// TIA Portal V16 export
// export: Created 2022-02-04T14:40:10.8066847Z, ExportSetting WithDefaults, DisplayName Totally Integrated Automation Portal, DisplayVersion V16 Update 1, DisplayName TIA Portal Version Control Interface, DisplayVersion V16, DisplayName TIA Portal Openness, DisplayVersion V16, DisplayName SINAMICS Startdrive Advanced, DisplayVersion V16 Update 5, DisplayName SINAMICS Startdrive G130, G150, S120, S150, SINAMICS MV, S210, DisplayVersion V16 Update 5, DisplayName SINAMICS Startdrive G110M, G120, G120C, G120D, G120P, G115D, DisplayVersion V16 Update 5, DisplayName STEP 7 Professional, DisplayVersion V16, DisplayName STEP 7 Safety, DisplayVersion V16, DisplayName WinCC Advanced, DisplayVersion V16, DisplayName SIMATIC Visualization Architect, DisplayVersion V16
FUNCTION_BLOCK "ПФМ Брака"   // FB3, LAD
VERSION : 0.1
// логика работы ПФМ брака
// stored: AutoNumber true, IsIECCheckEnabled false, UDAEnableTagReadback false
   VAR DB_SPECIFIC
      Trig332 : Bool;   // Тригер М332 сброс доски
      "TrigS79.3" : Bool;   // Тригер Авто режима
      ForcingPacket : Bool;
      LiftPushingPacket : Bool;   // лифт занят
      HodVil2 { ExternalAccessible := 'False'; ExternalVisible := 'False'; ExternalWritable := 'False'} : Bool;   // Триггер ход вил М335
      HodVil { ExternalAccessible := 'False'; ExternalVisible := 'False'; ExternalWritable := 'False'} : Bool;   // Триггер ход вил М335
      ForcingLift : Bool;
      CountSensor_front : Bool;
      StopDovod : Bool;
      StopDropppingBoards : Bool;
      newBob_old : Bool;
      liftDown_old : Bool;
      liftPushingPacket_old : Bool;
      newBoard_old : Bool;
      Upor_Off_trig : Bool;
      Lift_GoToStartPosition : Bool;
      ReviveSignal : Bool;   // сигнал для оживления механизмов
      StartAwaitForGasket : Bool;   // ожидание прокладок
      AwaitGasket : Bool;
      AlarmNotReadedPack : Bool;
      AlarmExtraBoardInLay : Bool;   // авария лишняя доска на слой ПФМ брака
      AlarmNoPacketPushed : Bool;
      BoardsInLayCounter : Int;   // Сравнение счетчика 2
      LayersCounter : Int;   // Счет слоев досок
   END_VAR
   VAR
      Board_counter : "Adder";   // Счетчик досок в слое
      Lay_counter : "Adder";   // Счетчик слоев
   END_VAR
   VAR_TEMP
      start_await : Bool;
      Sert : Word;
   END_VAR
   VAR_TEMP   // added for the SCL form of the ladder/FBD networks
      _w1 : Bool;
      _w2 : Bool;
      _w3 : Bool;
      _s5time1 : S5Time;
   END_VAR
BEGIN

REGION Network 1: Реле безопасности К41 группа 331,332-337
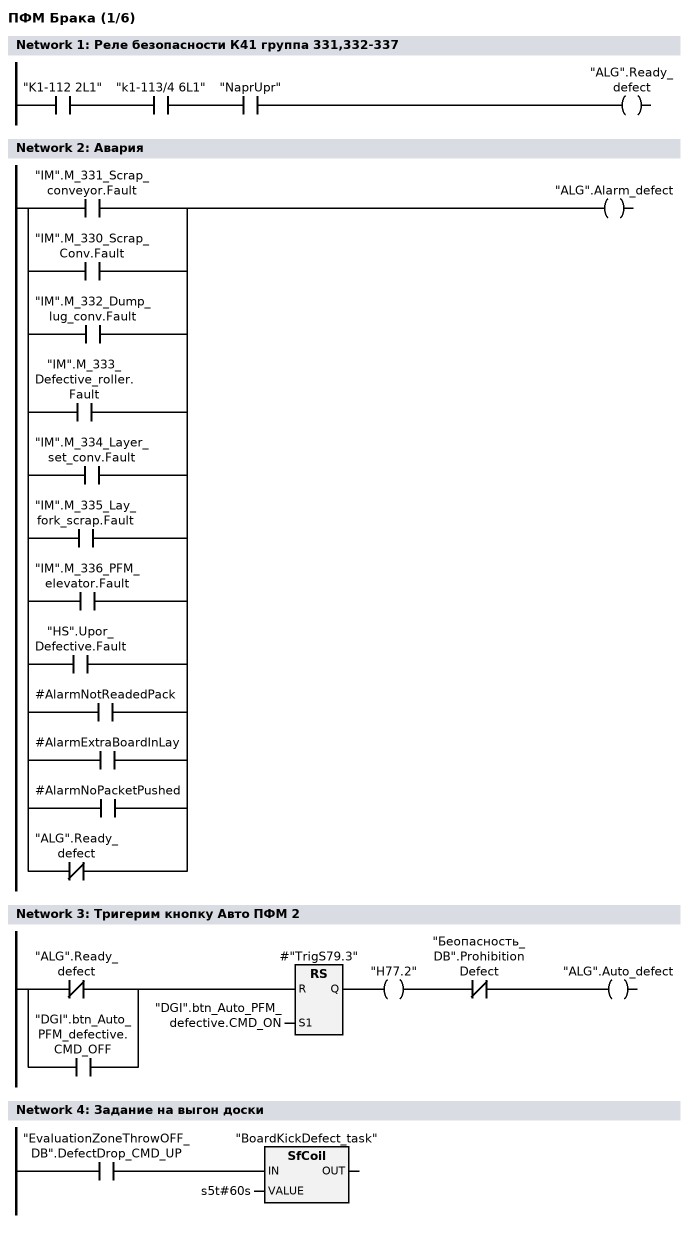
   RUNG wire#powerrail
      Contact( "K1-112 2L1" )
      Contact( "k1-113/4 6L1" )
      Contact( "NaprUpr" )
      Coil( "ALG".Ready_defect )
   END_RUNG
   // the same network as SCL:
   "ALG".Ready_defect := "K1-112 2L1" AND "k1-113/4 6L1" AND "NaprUpr";
END_REGION

REGION Network 2: Авария
   RUNG wire#powerrail
      Contact( "IM".M_331_Scrap_conveyor.Fault )
      wire#w1
      Coil( "ALG".Alarm_defect )
   END_RUNG
   RUNG wire#powerrail
      Contact( "IM".M_330_Scrap_Conv.Fault )
   END_RUNG wire#w1
   RUNG wire#powerrail
      Contact( "IM".M_332_Dump_lug_conv.Fault )
   END_RUNG wire#w1
   RUNG wire#powerrail
      Contact( "IM".M_333_Defective_roller.Fault )
   END_RUNG wire#w1
   RUNG wire#powerrail
      Contact( "IM".M_334_Layer_set_conv.Fault )
   END_RUNG wire#w1
   RUNG wire#powerrail
      Contact( "IM".M_335_Lay_fork_scrap.Fault )
   END_RUNG wire#w1
   RUNG wire#powerrail
      Contact( "IM".M_336_PFM_elevator.Fault )
   END_RUNG wire#w1
   RUNG wire#powerrail
      Contact( "HS".Upor_Defective.Fault )
   END_RUNG wire#w1
   RUNG wire#powerrail
      Contact( #AlarmNotReadedPack )
   END_RUNG wire#w1
   RUNG wire#powerrail
      Contact( #AlarmExtraBoardInLay )
   END_RUNG wire#w1
   RUNG wire#powerrail
      Contact( #AlarmNoPacketPushed )
   END_RUNG wire#w1
   RUNG wire#powerrail
      I_Contact( "ALG".Ready_defect )
   END_RUNG wire#w1
   // the same network as SCL:
   "ALG".Alarm_defect := "IM".M_331_Scrap_conveyor.Fault OR "IM".M_330_Scrap_Conv.Fault OR "IM".M_332_Dump_lug_conv.Fault OR "IM".M_333_Defective_roller.Fault OR "IM".M_334_Layer_set_conv.Fault OR "IM".M_335_Lay_fork_scrap.Fault OR "IM".M_336_PFM_elevator.Fault OR "HS".Upor_Defective.Fault OR #AlarmNotReadedPack OR #AlarmExtraBoardInLay OR #AlarmNoPacketPushed OR NOT "ALG".Ready_defect;
END_REGION

REGION Network 3: Тригерим кнопку Авто ПФМ 2
   RUNG wire#powerrail
      I_Contact( "ALG".Ready_defect )
      wire#w1
      S_RS(operand := #"TrigS79.3", s1 := "DGI".btn_Auto_PFM_defective.CMD_ON)
      Coil( "H77.2" )
      I_Contact( "Беопасность_DB".ProhibitionDefect )
      Coil( "ALG".Auto_defect )
   END_RUNG
   RUNG wire#powerrail
      Contact( "DGI".btn_Auto_PFM_defective.CMD_OFF )
   END_RUNG wire#w1
   // the same network as SCL:
   IF NOT "ALG".Ready_defect OR "DGI".btn_Auto_PFM_defective.CMD_OFF THEN
       #"TrigS79.3" := FALSE;   // RS flip-flop
   END_IF;
   IF "DGI".btn_Auto_PFM_defective.CMD_ON THEN #"TrigS79.3" := TRUE; END_IF;
   "H77.2" := #"TrigS79.3";
   "ALG".Auto_defect := #"TrigS79.3" AND NOT "Беопасность_DB".ProhibitionDefect;
END_REGION

REGION Network 4: Задание на выгон доски
   // no SCL statement known for SfCoil: written as a call
   SfCoil(in := "EvaluationZoneThrowOFF_DB".DefectDrop_CMD_UP,
          value := s5t#60s,
          operand := "BoardKickDefect_task");
END_REGION

REGION Network 5: Авто вперед М331/ M330
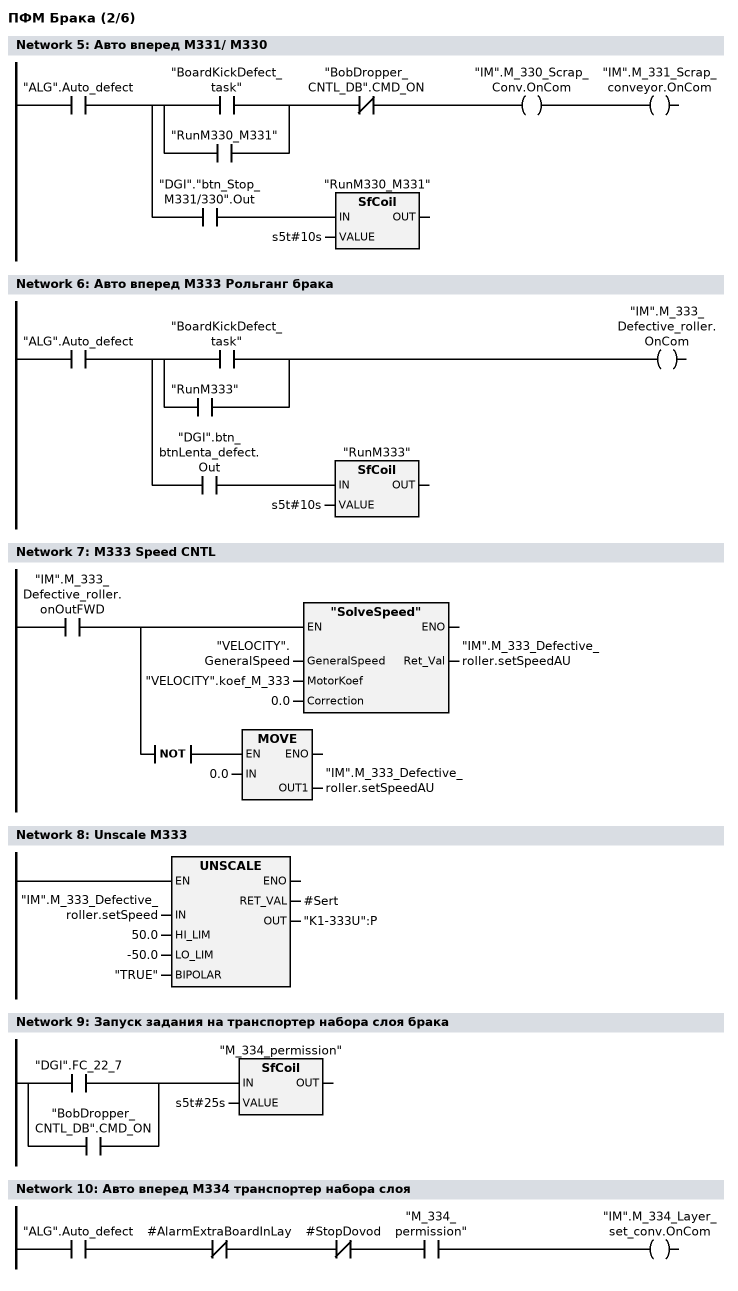
   // no SCL statement known for SfCoil: written as a call
   "IM".M_330_Scrap_Conv.OnCom := "ALG".Auto_defect AND ("BoardKickDefect_task" OR "RunM330_M331") AND NOT "BobDropper_CNTL_DB".CMD_ON;
   "IM".M_331_Scrap_conveyor.OnCom := "IM".M_330_Scrap_Conv.OnCom;
   SfCoil(in := "ALG".Auto_defect AND "DGI"."btn_Stop_M331/330".Out,
          value := s5t#10s,
          operand := "RunM330_M331");
END_REGION

REGION Network 6: Авто вперед М333 Рольганг брака
   // no SCL statement known for SfCoil: written as a call
   "IM".M_333_Defective_roller.OnCom := "ALG".Auto_defect AND ("BoardKickDefect_task" OR "RunM333");
   SfCoil(in := "ALG".Auto_defect AND "DGI".btn_btnLenta_defect.Out, value := s5t#10s, operand := "RunM333");
END_REGION

REGION Network 7: М333 Speed CNTL
   RUNG wire#powerrail
      Contact( "IM".M_333_Defective_roller.onOutFWD )
      wire#w1
      "SolveSpeed"(GeneralSpeed := "VELOCITY".GeneralSpeed, MotorKoef := "VELOCITY".koef_M_333, Correction := 0.0, Ret_Val => "IM".M_333_Defective_roller.setSpeedAU)
   END_RUNG
   RUNG wire#w1
      Not()
      { S7_GenerateENO := "TRUE" } Move(in := 0.0, out1 => "IM".M_333_Defective_roller.setSpeedAU)
   END_RUNG
   // the same network as SCL:
   #_w1 := "IM".M_333_Defective_roller.onOutFWD;
   IF #_w1 THEN
       "IM".M_333_Defective_roller.setSpeedAU := "SolveSpeed"(GeneralSpeed := "VELOCITY".GeneralSpeed,
                               MotorKoef := "VELOCITY".koef_M_333,
                               Correction := 0.0);
   END_IF;
   IF NOT #_w1 THEN "IM".M_333_Defective_roller.setSpeedAU := 0.0; END_IF;
END_REGION

REGION Network 8: Unscale M333
   RUNG wire#powerrail
      UNSCALE(IN := "IM".M_333_Defective_roller.setSpeed, HI_LIM := 50.0, LO_LIM := -50.0, BIPOLAR := "TRUE", RET_VAL => #Sert, OUT => "K1-333U":P)
   END_RUNG
   // the same network as SCL:
   #Sert := UNSCALE(IN := "IM".M_333_Defective_roller.setSpeed,
                    HI_LIM := 50.0,
                    LO_LIM := -50.0,
                    BIPOLAR := "TRUE",
                    OUT => "K1-333U":P);
END_REGION

REGION Network 9: Запуск задания на транспортер набора слоя брака
   // no SCL statement known for SfCoil: written as a call
   SfCoil(in := "DGI".FC_22_7 OR "BobDropper_CNTL_DB".CMD_ON, value := s5t#25s, operand := "M_334_permission");
END_REGION

REGION Network 10: Авто вперед М334 транспортер набора слоя
   RUNG wire#powerrail
      Contact( "ALG".Auto_defect )
      I_Contact( #AlarmExtraBoardInLay )
      I_Contact( #StopDovod )
      Contact( "M_334_permission" )
      Coil( "IM".M_334_Layer_set_conv.OnCom )
   END_RUNG
   // the same network as SCL:
   "IM".M_334_Layer_set_conv.OnCom := "ALG".Auto_defect AND NOT #AlarmExtraBoardInLay AND NOT #StopDovod AND "M_334_permission";
END_REGION

REGION Network 11: М334 транспортер набора слоя команды на движение
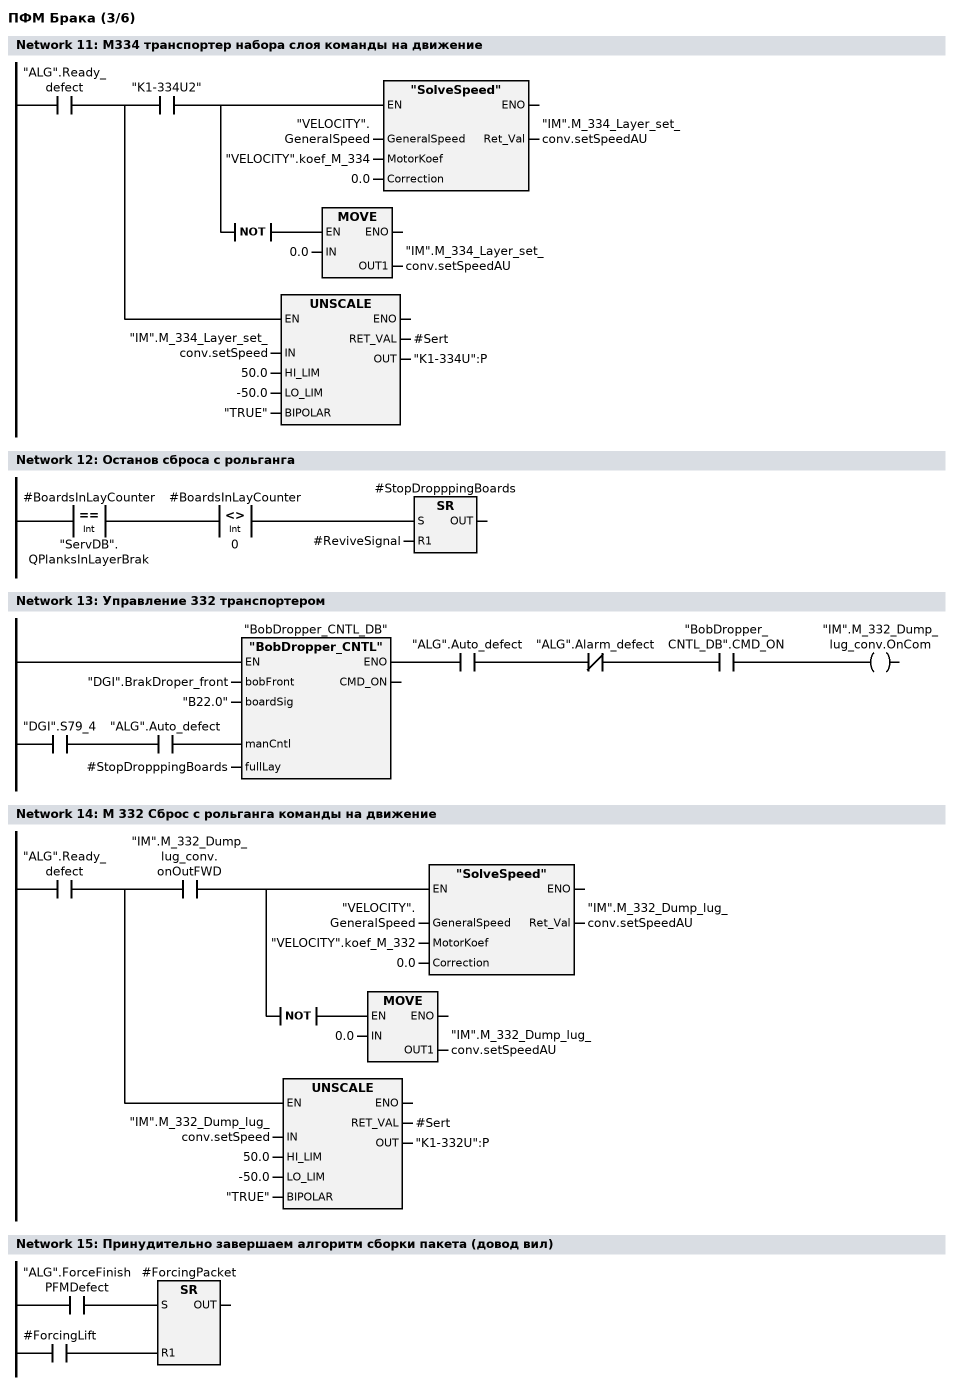
   RUNG wire#powerrail
      Contact( "ALG".Ready_defect )
      wire#w1
      Contact( "K1-334U2" )
      wire#w2
      "SolveSpeed"(GeneralSpeed := "VELOCITY".GeneralSpeed, MotorKoef := "VELOCITY".koef_M_334, Correction := 0.0, Ret_Val => "IM".M_334_Layer_set_conv.setSpeedAU)
   END_RUNG
   RUNG wire#w2
      Not()
      { S7_GenerateENO := "TRUE" } Move(in := 0.0, out1 => "IM".M_334_Layer_set_conv.setSpeedAU)
   END_RUNG
   RUNG wire#w1
      UNSCALE(IN := "IM".M_334_Layer_set_conv.setSpeed, HI_LIM := 50.0, LO_LIM := -50.0, BIPOLAR := "TRUE", RET_VAL => #Sert, OUT => "K1-334U":P)
   END_RUNG
   // the same network as SCL:
   #_w1 := "ALG".Ready_defect AND "K1-334U2";
   #_w2 := "ALG".Ready_defect;
   IF #_w1 THEN
       "IM".M_334_Layer_set_conv.setSpeedAU := "SolveSpeed"(GeneralSpeed := "VELOCITY".GeneralSpeed,
                               MotorKoef := "VELOCITY".koef_M_334,
                               Correction := 0.0);
   END_IF;
   IF NOT #_w1 THEN "IM".M_334_Layer_set_conv.setSpeedAU := 0.0; END_IF;
   IF #_w2 THEN
       #Sert := UNSCALE(IN := "IM".M_334_Layer_set_conv.setSpeed,
                        HI_LIM := 50.0,
                        LO_LIM := -50.0,
                        BIPOLAR := "TRUE",
                        OUT => "K1-334U":P);
   END_IF;
END_REGION

REGION Network 12: Останов сброса с рольганга
   RUNG wire#powerrail
      { S7_Templates := "SrcType := Int" } EQ_Contact(in1 := #BoardsInLayCounter, in2 := "ServDB".QPlanksInLayerBrak)
      { S7_Templates := "SrcType := Int" } NE_Contact(in1 := #BoardsInLayCounter, in2 := 0)
      S_SR(operand := #StopDropppingBoards, r1 := #ReviveSignal)
   END_RUNG
   // the same network as SCL:
   IF (#BoardsInLayCounter = "ServDB".QPlanksInLayerBrak) AND (#BoardsInLayCounter <> 0) THEN
       #StopDropppingBoards := TRUE;   // SR flip-flop
   END_IF;
   IF #ReviveSignal THEN #StopDropppingBoards := FALSE; END_IF;
END_REGION

REGION Network 13: Управление 332 транспортером
   RUNG wire#powerrail
      "BobDropper_CNTL_DB"(manCntl := wire#w1, bobFront := "DGI".BrakDroper_front, boardSig := "B22.0", fullLay := #StopDropppingBoards, CMD_ON =>)
      Contact( "ALG".Auto_defect )
      I_Contact( "ALG".Alarm_defect )
      Contact( "BobDropper_CNTL_DB".CMD_ON )
      Coil( "IM".M_332_Dump_lug_conv.OnCom )
   END_RUNG
   RUNG wire#powerrail
      Contact( "DGI".S79_4 )
      Contact( "ALG".Auto_defect )
   END_RUNG wire#w1
   // the same network as SCL:
   "BobDropper_CNTL_DB"(bobFront := "DGI".BrakDroper_front,   // "BobDropper_CNTL"
                        boardSig := "B22.0",
                        manCntl := "DGI".S79_4 AND "ALG".Auto_defect,
                        fullLay := #StopDropppingBoards,
                        ENO => #_w1);
   "IM".M_332_Dump_lug_conv.OnCom := #_w1 AND "ALG".Auto_defect AND NOT "ALG".Alarm_defect AND "BobDropper_CNTL_DB".CMD_ON;
END_REGION

REGION Network 14: М 332 Сброс с рольганга команды на движение
   RUNG wire#powerrail
      Contact( "ALG".Ready_defect )
      wire#w1
      Contact( "IM".M_332_Dump_lug_conv.onOutFWD )
      wire#w2
      "SolveSpeed"(GeneralSpeed := "VELOCITY".GeneralSpeed, MotorKoef := "VELOCITY".koef_M_332, Correction := 0.0, Ret_Val => "IM".M_332_Dump_lug_conv.setSpeedAU)
   END_RUNG
   RUNG wire#w2
      Not()
      { S7_GenerateENO := "TRUE" } Move(in := 0.0, out1 => "IM".M_332_Dump_lug_conv.setSpeedAU)
   END_RUNG
   RUNG wire#w1
      UNSCALE(IN := "IM".M_332_Dump_lug_conv.setSpeed, HI_LIM := 50.0, LO_LIM := -50.0, BIPOLAR := "TRUE", RET_VAL => #Sert, OUT => "K1-332U":P)
   END_RUNG
   // the same network as SCL:
   #_w1 := "ALG".Ready_defect AND "IM".M_332_Dump_lug_conv.onOutFWD;
   #_w2 := "ALG".Ready_defect;
   IF #_w1 THEN
       "IM".M_332_Dump_lug_conv.setSpeedAU := "SolveSpeed"(GeneralSpeed := "VELOCITY".GeneralSpeed,
                               MotorKoef := "VELOCITY".koef_M_332,
                               Correction := 0.0);
   END_IF;
   IF NOT #_w1 THEN "IM".M_332_Dump_lug_conv.setSpeedAU := 0.0; END_IF;
   IF #_w2 THEN
       #Sert := UNSCALE(IN := "IM".M_332_Dump_lug_conv.setSpeed,
                        HI_LIM := 50.0,
                        LO_LIM := -50.0,
                        BIPOLAR := "TRUE",
                        OUT => "K1-332U":P);
   END_IF;
END_REGION

REGION Network 15: Принудительно завершаем алгоритм сборки пакета (довод вил)
   RUNG wire#powerrail
      Contact( "ALG".ForceFinishPFMDefect )
      S_SR(operand := #ForcingPacket, r1 := wire#w1)
   END_RUNG
   RUNG wire#powerrail
      Contact( #ForcingLift )
   END_RUNG wire#w1
   // the same network as SCL:
   IF "ALG".ForceFinishPFMDefect THEN
       #ForcingPacket := TRUE;   // SR flip-flop
   END_IF;
   IF #ForcingLift THEN #ForcingPacket := FALSE; END_IF;
END_REGION

REGION Network 16: Форсирование сборки пакета ПФМ (лифт)
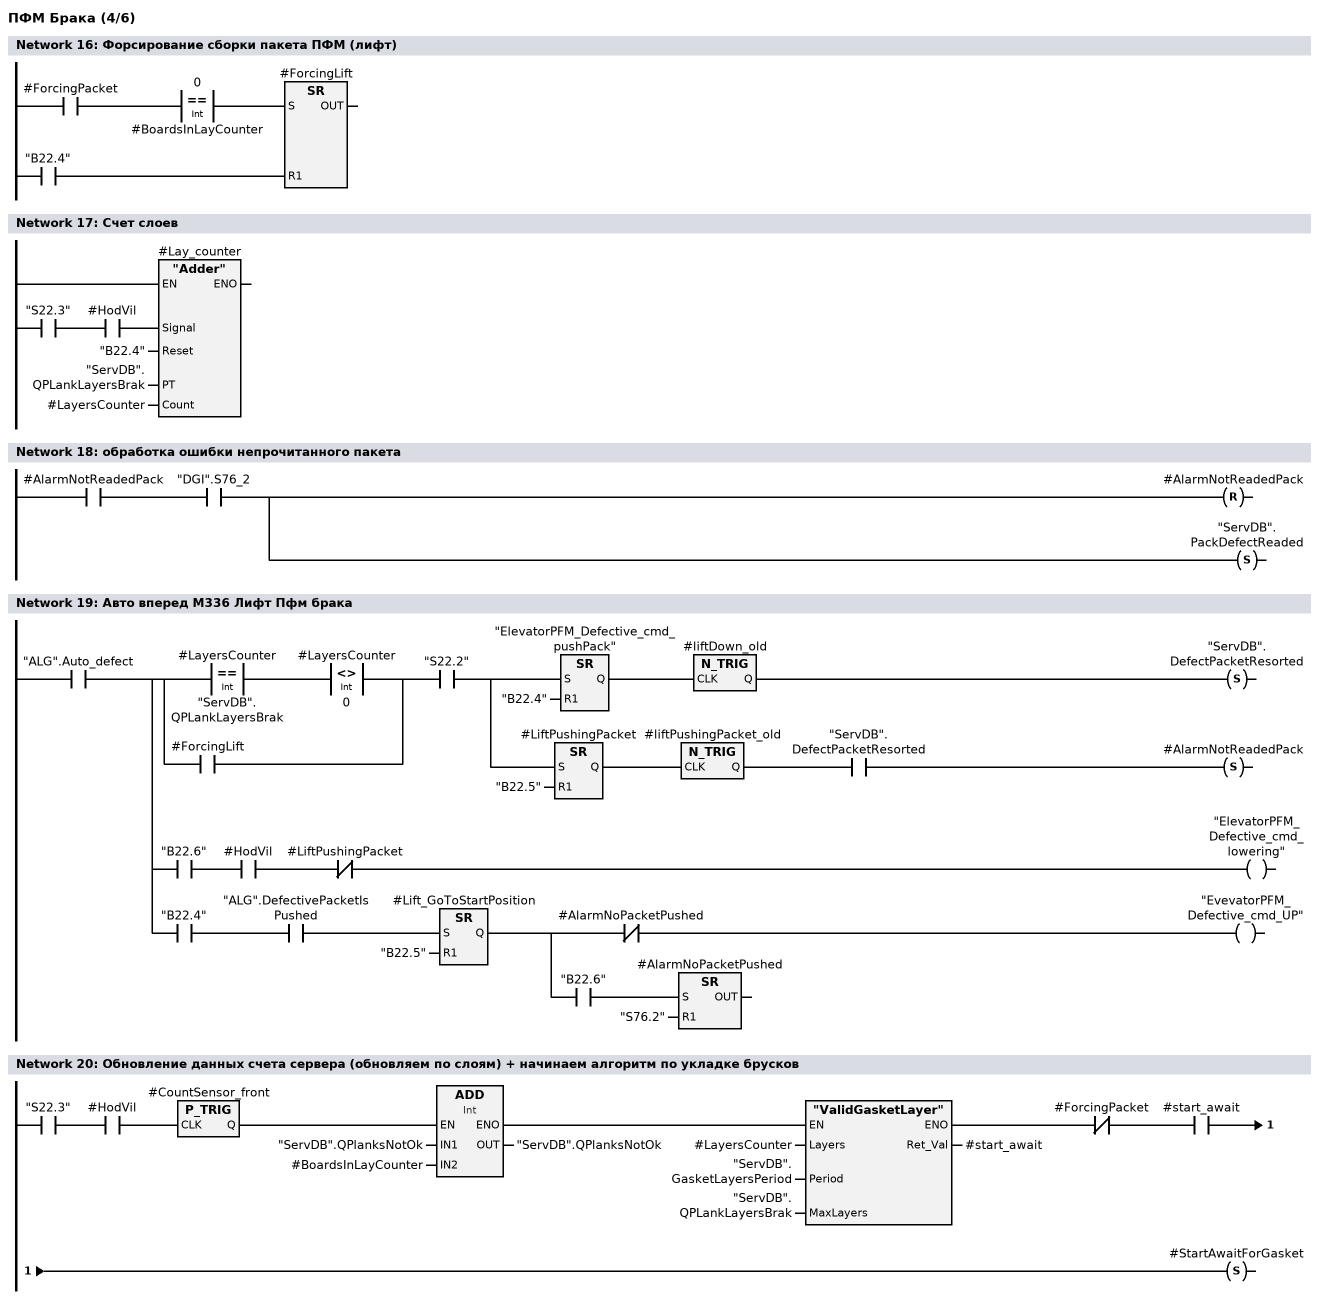
   RUNG wire#powerrail
      Contact( #ForcingPacket )
      { S7_Templates := "SrcType := Int" } EQ_Contact(in1 := 0, in2 := #BoardsInLayCounter)
      S_SR(operand := #ForcingLift, r1 := wire#w1)
   END_RUNG
   RUNG wire#powerrail
      Contact( "B22.4" )
   END_RUNG wire#w1
   // the same network as SCL:
   IF #ForcingPacket AND (0 = #BoardsInLayCounter) THEN
       #ForcingLift := TRUE;   // SR flip-flop
   END_IF;
   IF "B22.4" THEN #ForcingLift := FALSE; END_IF;
END_REGION

REGION Network 17: Счет слоев
   RUNG wire#powerrail
      #Lay_counter(Signal := wire#w1, Reset := "B22.4", PT := "ServDB".QPLankLayersBrak, Count := #LayersCounter)
   END_RUNG
   RUNG wire#powerrail
      Contact( "S22.3" )
      Contact( #HodVil )
   END_RUNG wire#w1
   // the same network as SCL:
   #Lay_counter(Signal := "S22.3" AND #HodVil,   // "Adder"
                Reset := "B22.4",
                PT := "ServDB".QPLankLayersBrak,
                Count := #LayersCounter);
END_REGION

REGION Network 18: обработка ошибки непрочитанного пакета
   RUNG wire#powerrail
      Contact( #AlarmNotReadedPack )
      Contact( "DGI".S76_2 )
      wire#w1
      R_Coil( #AlarmNotReadedPack )
   END_RUNG
   RUNG wire#w1
      S_Coil( "ServDB".PackDefectReaded )
   END_RUNG
   // the same network as SCL:
   #_w1 := #AlarmNotReadedPack AND "DGI".S76_2;
   IF #_w1 THEN
       #AlarmNotReadedPack := FALSE;
       "ServDB".PackDefectReaded := TRUE;
   END_IF;
END_REGION

REGION Network 19: Авто вперед М336 Лифт Пфм брака
   RUNG wire#powerrail
      Contact( "ALG".Auto_defect )
      wire#w1
      { S7_Templates := "SrcType := Int" } EQ_Contact(in1 := #LayersCounter, in2 := "ServDB".QPLankLayersBrak)
      { S7_Templates := "SrcType := Int" } NE_Contact(in1 := #LayersCounter, in2 := 0)
      wire#w2
      Contact( "S22.2" )
      wire#w3
      S_SR(operand := "ElevatorPFM_Defective_cmd_pushPack", r1 := "B22.4")
      N_Trig( #liftDown_old )
      S_Coil( "ServDB".DefectPacketResorted )
   END_RUNG
   RUNG wire#w1
      Contact( #ForcingLift )
   END_RUNG wire#w2
   RUNG wire#w3
      S_SR(operand := #LiftPushingPacket, r1 := "B22.5")
      N_Trig( #liftPushingPacket_old )
      Contact( "ServDB".DefectPacketResorted )
      S_Coil( #AlarmNotReadedPack )
   END_RUNG
   RUNG wire#w1
      Contact( "B22.6" )
      Contact( #HodVil )
      I_Contact( #LiftPushingPacket )
      Coil( "ElevatorPFM_Defective_cmd_lowering" )
   END_RUNG
   RUNG wire#w1
      Contact( "B22.4" )
      Contact( "ALG".DefectivePacketIsPushed )
      S_SR(operand := #Lift_GoToStartPosition, r1 := "B22.5")
      wire#w4
      I_Contact( #AlarmNoPacketPushed )
      Coil( "EvevatorPFM_Defective_cmd_UP" )
   END_RUNG
   RUNG wire#w4
      Contact( "B22.6" )
      S_SR(operand := #AlarmNoPacketPushed, r1 := "S76.2")
   END_RUNG
   // the same network as SCL:
   #_w1 := "ALG".Auto_defect AND (((#LayersCounter = "ServDB".QPLankLayersBrak) AND (#LayersCounter <> 0)) OR #ForcingLift) AND "S22.2";
   IF #_w1 THEN
       "ElevatorPFM_Defective_cmd_pushPack" := TRUE;   // SR flip-flop
   END_IF;
   IF "B22.4" THEN "ElevatorPFM_Defective_cmd_pushPack" := FALSE; END_IF;
   #_w2 := NOT "ElevatorPFM_Defective_cmd_pushPack" AND #liftDown_old;   // falling edge
   #liftDown_old := "ElevatorPFM_Defective_cmd_pushPack";
   IF #_w2 THEN "ServDB".DefectPacketResorted := TRUE; END_IF;
   IF #_w1 THEN
       #LiftPushingPacket := TRUE;   // SR flip-flop
   END_IF;
   IF "B22.5" THEN #LiftPushingPacket := FALSE; END_IF;
   #_w3 := NOT #LiftPushingPacket AND #liftPushingPacket_old;   // falling edge
   #liftPushingPacket_old := #LiftPushingPacket;
   IF #_w3 AND "ServDB".DefectPacketResorted THEN #AlarmNotReadedPack := TRUE; END_IF;
   "ElevatorPFM_Defective_cmd_lowering" := "ALG".Auto_defect AND "B22.6" AND #HodVil AND NOT #LiftPushingPacket;
   IF "ALG".Auto_defect AND "B22.4" AND "ALG".DefectivePacketIsPushed THEN
       #Lift_GoToStartPosition := TRUE;   // SR flip-flop
   END_IF;
   IF "B22.5" THEN #Lift_GoToStartPosition := FALSE; END_IF;
   "EvevatorPFM_Defective_cmd_UP" := #Lift_GoToStartPosition AND NOT #AlarmNoPacketPushed;
   IF #Lift_GoToStartPosition AND "B22.6" THEN
       #AlarmNoPacketPushed := TRUE;   // SR flip-flop
   END_IF;
   IF "S76.2" THEN #AlarmNoPacketPushed := FALSE; END_IF;
END_REGION

REGION Network 20: Обновление данных счета сервера (обновляем по слоям) + начинаем алгоритм по укладке брусков
   RUNG wire#powerrail
      Contact( "S22.3" )
      Contact( #HodVil )
      P_Trig( #CountSensor_front )
      { S7_Templates := "SrcType := Int"; S7_GenerateENO := "TRUE" } Add(in1 := "ServDB".QPlanksNotOk, in2 := #BoardsInLayCounter, out => "ServDB".QPlanksNotOk)
      "ValidGasketLayer"(Layers := #LayersCounter, Period := "ServDB".GasketLayersPeriod, MaxLayers := "ServDB".QPLankLayersBrak, Ret_Val => #start_await)
      I_Contact( #ForcingPacket )
      Contact( #start_await )
      S_Coil( #StartAwaitForGasket )
   END_RUNG
   // the same network as SCL:
   // ENO of a box is taken as its EN; it also drops when the box reports an error
   #_w1 := "S22.3" AND #HodVil;
   #_w2 := #_w1 AND NOT #CountSensor_front;   // rising edge
   #CountSensor_front := #_w1;
   IF #_w2 THEN "ServDB".QPlanksNotOk := "ServDB".QPlanksNotOk + #BoardsInLayCounter; END_IF;
   #start_await := "ValidGasketLayer"(EN := #_w2,
                           Layers := #LayersCounter,
                           Period := "ServDB".GasketLayersPeriod,
                           MaxLayers := "ServDB".QPLankLayersBrak,
                           ENO => #_w3);
   IF #_w3 AND NOT #ForcingPacket AND #start_await THEN #StartAwaitForGasket := TRUE; END_IF;
END_REGION

REGION Network 21: Логика ожидания уложенных прокладок на пакет Брака
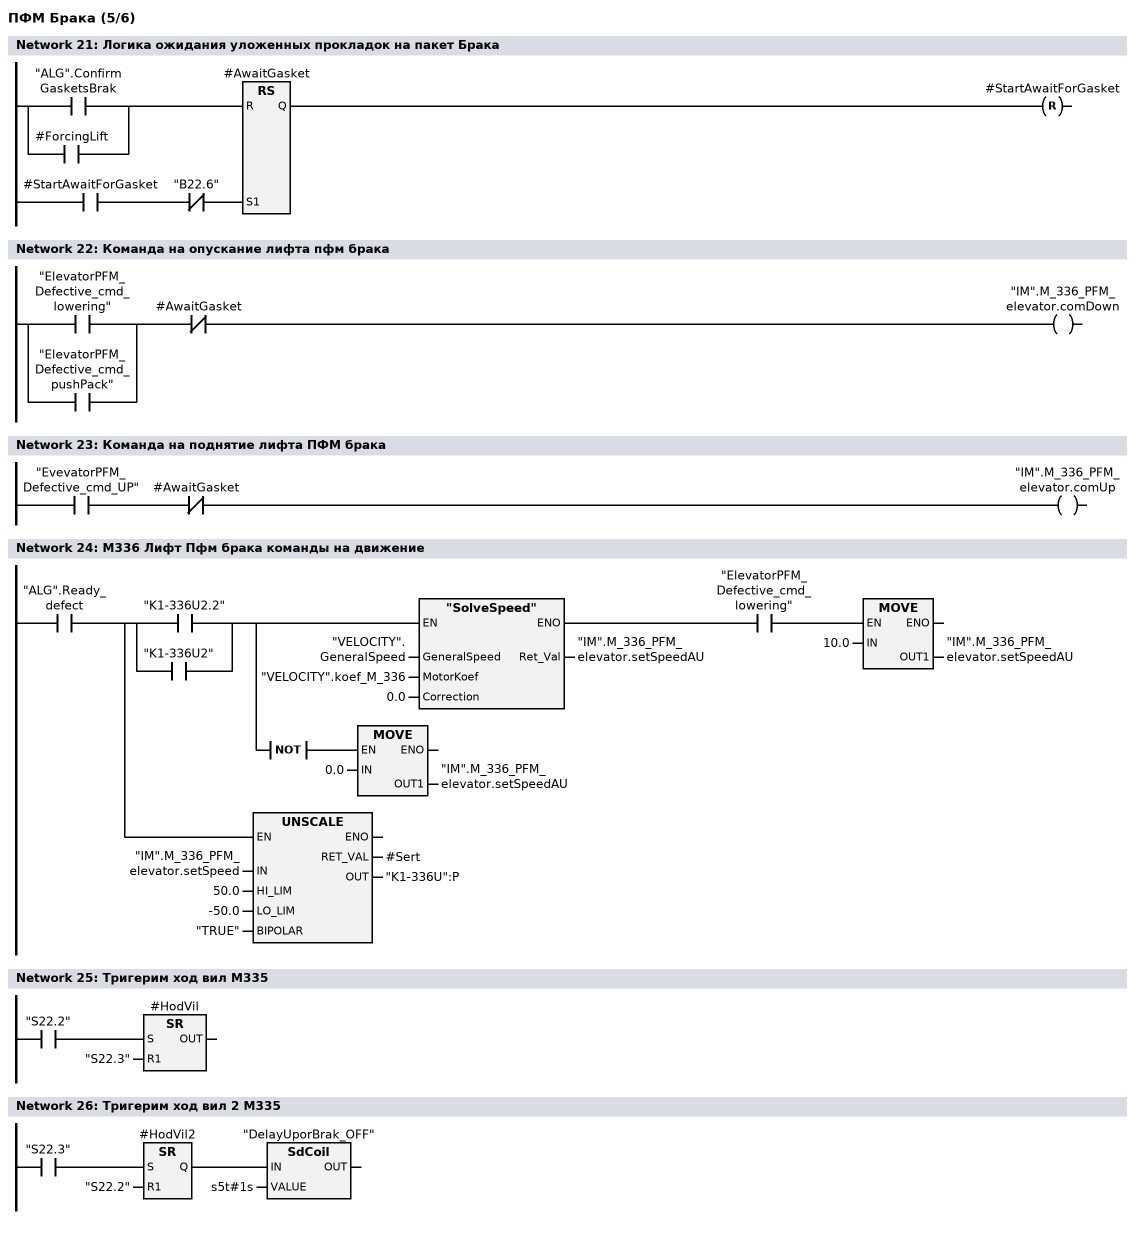
   RUNG wire#powerrail
      Contact( "ALG".ConfirmGasketsBrak )
      wire#w1
      S_RS(operand := #AwaitGasket, s1 := wire#w2)
      R_Coil( #StartAwaitForGasket )
   END_RUNG
   RUNG wire#powerrail
      Contact( #ForcingLift )
   END_RUNG wire#w1
   RUNG wire#powerrail
      Contact( #StartAwaitForGasket )
      I_Contact( "B22.6" )
   END_RUNG wire#w2
   // the same network as SCL:
   IF "ALG".ConfirmGasketsBrak OR #ForcingLift THEN
       #AwaitGasket := FALSE;   // RS flip-flop
   END_IF;
   IF #StartAwaitForGasket AND NOT "B22.6" THEN #AwaitGasket := TRUE; END_IF;
   IF #AwaitGasket THEN #StartAwaitForGasket := FALSE; END_IF;
END_REGION

REGION Network 22: Команда на опускание лифта пфм брака
   RUNG wire#powerrail
      Contact( "ElevatorPFM_Defective_cmd_lowering" )
      wire#w1
      I_Contact( #AwaitGasket )
      Coil( "IM".M_336_PFM_elevator.comDown )
   END_RUNG
   RUNG wire#powerrail
      Contact( "ElevatorPFM_Defective_cmd_pushPack" )
   END_RUNG wire#w1
   // the same network as SCL:
   "IM".M_336_PFM_elevator.comDown := ("ElevatorPFM_Defective_cmd_lowering" OR "ElevatorPFM_Defective_cmd_pushPack") AND NOT #AwaitGasket;
END_REGION

REGION Network 23: Команда на поднятие лифта ПФМ брака
   RUNG wire#powerrail
      Contact( "EvevatorPFM_Defective_cmd_UP" )
      I_Contact( #AwaitGasket )
      Coil( "IM".M_336_PFM_elevator.comUp )
   END_RUNG
   // the same network as SCL:
   "IM".M_336_PFM_elevator.comUp := "EvevatorPFM_Defective_cmd_UP" AND NOT #AwaitGasket;
END_REGION

REGION Network 24: М336 Лифт Пфм брака команды на движение
   RUNG wire#powerrail
      Contact( "ALG".Ready_defect )
      wire#w1
      Contact( "K1-336U2.2" )
      wire#w2
      "SolveSpeed"(GeneralSpeed := "VELOCITY".GeneralSpeed, MotorKoef := "VELOCITY".koef_M_336, Correction := 0.0, Ret_Val => "IM".M_336_PFM_elevator.setSpeedAU)
      Contact( "ElevatorPFM_Defective_cmd_lowering" )
      { S7_GenerateENO := "TRUE" } Move(in := 10.0, out1 => "IM".M_336_PFM_elevator.setSpeedAU)
   END_RUNG
   RUNG wire#w1
      Contact( "K1-336U2" )
   END_RUNG wire#w2
   RUNG wire#w2
      Not()
      { S7_GenerateENO := "TRUE" } Move(in := 0.0, out1 => "IM".M_336_PFM_elevator.setSpeedAU)
   END_RUNG
   RUNG wire#w1
      UNSCALE(IN := "IM".M_336_PFM_elevator.setSpeed, HI_LIM := 50.0, LO_LIM := -50.0, BIPOLAR := "TRUE", RET_VAL => #Sert, OUT => "K1-336U":P)
   END_RUNG
   // the same network as SCL:
   #_w1 := "ALG".Ready_defect AND ("K1-336U2.2" OR "K1-336U2");
   #_w3 := "ALG".Ready_defect;
   "IM".M_336_PFM_elevator.setSpeedAU := "SolveSpeed"(EN := #_w1,
                           GeneralSpeed := "VELOCITY".GeneralSpeed,
                           MotorKoef := "VELOCITY".koef_M_336,
                           Correction := 0.0,
                           ENO => #_w2);
   IF #_w2 AND "ElevatorPFM_Defective_cmd_lowering" THEN "IM".M_336_PFM_elevator.setSpeedAU := 10.0; END_IF;
   IF NOT #_w1 THEN "IM".M_336_PFM_elevator.setSpeedAU := 0.0; END_IF;
   IF #_w3 THEN
       #Sert := UNSCALE(IN := "IM".M_336_PFM_elevator.setSpeed,
                        HI_LIM := 50.0,
                        LO_LIM := -50.0,
                        BIPOLAR := "TRUE",
                        OUT => "K1-336U":P);
   END_IF;
END_REGION

REGION Network 25: Тригерим ход вил М335
   RUNG wire#powerrail
      Contact( "S22.2" )
      S_SR(operand := #HodVil, r1 := "S22.3")
   END_RUNG
   // the same network as SCL:
   IF "S22.2" THEN
       #HodVil := TRUE;   // SR flip-flop
   END_IF;
   IF "S22.3" THEN #HodVil := FALSE; END_IF;
END_REGION

REGION Network 26: Тригерим ход вил 2 М335
   // no SCL statement known for SdCoil: written as a call
   IF "S22.3" THEN
       #HodVil2 := TRUE;   // SR flip-flop
   END_IF;
   IF "S22.2" THEN #HodVil2 := FALSE; END_IF;
   SdCoil(in := #HodVil2, value := s5t#1s, operand := "DelayUporBrak_OFF");
END_REGION

REGION Network 27: авария убрать лишнюю доску с ПФМ брака
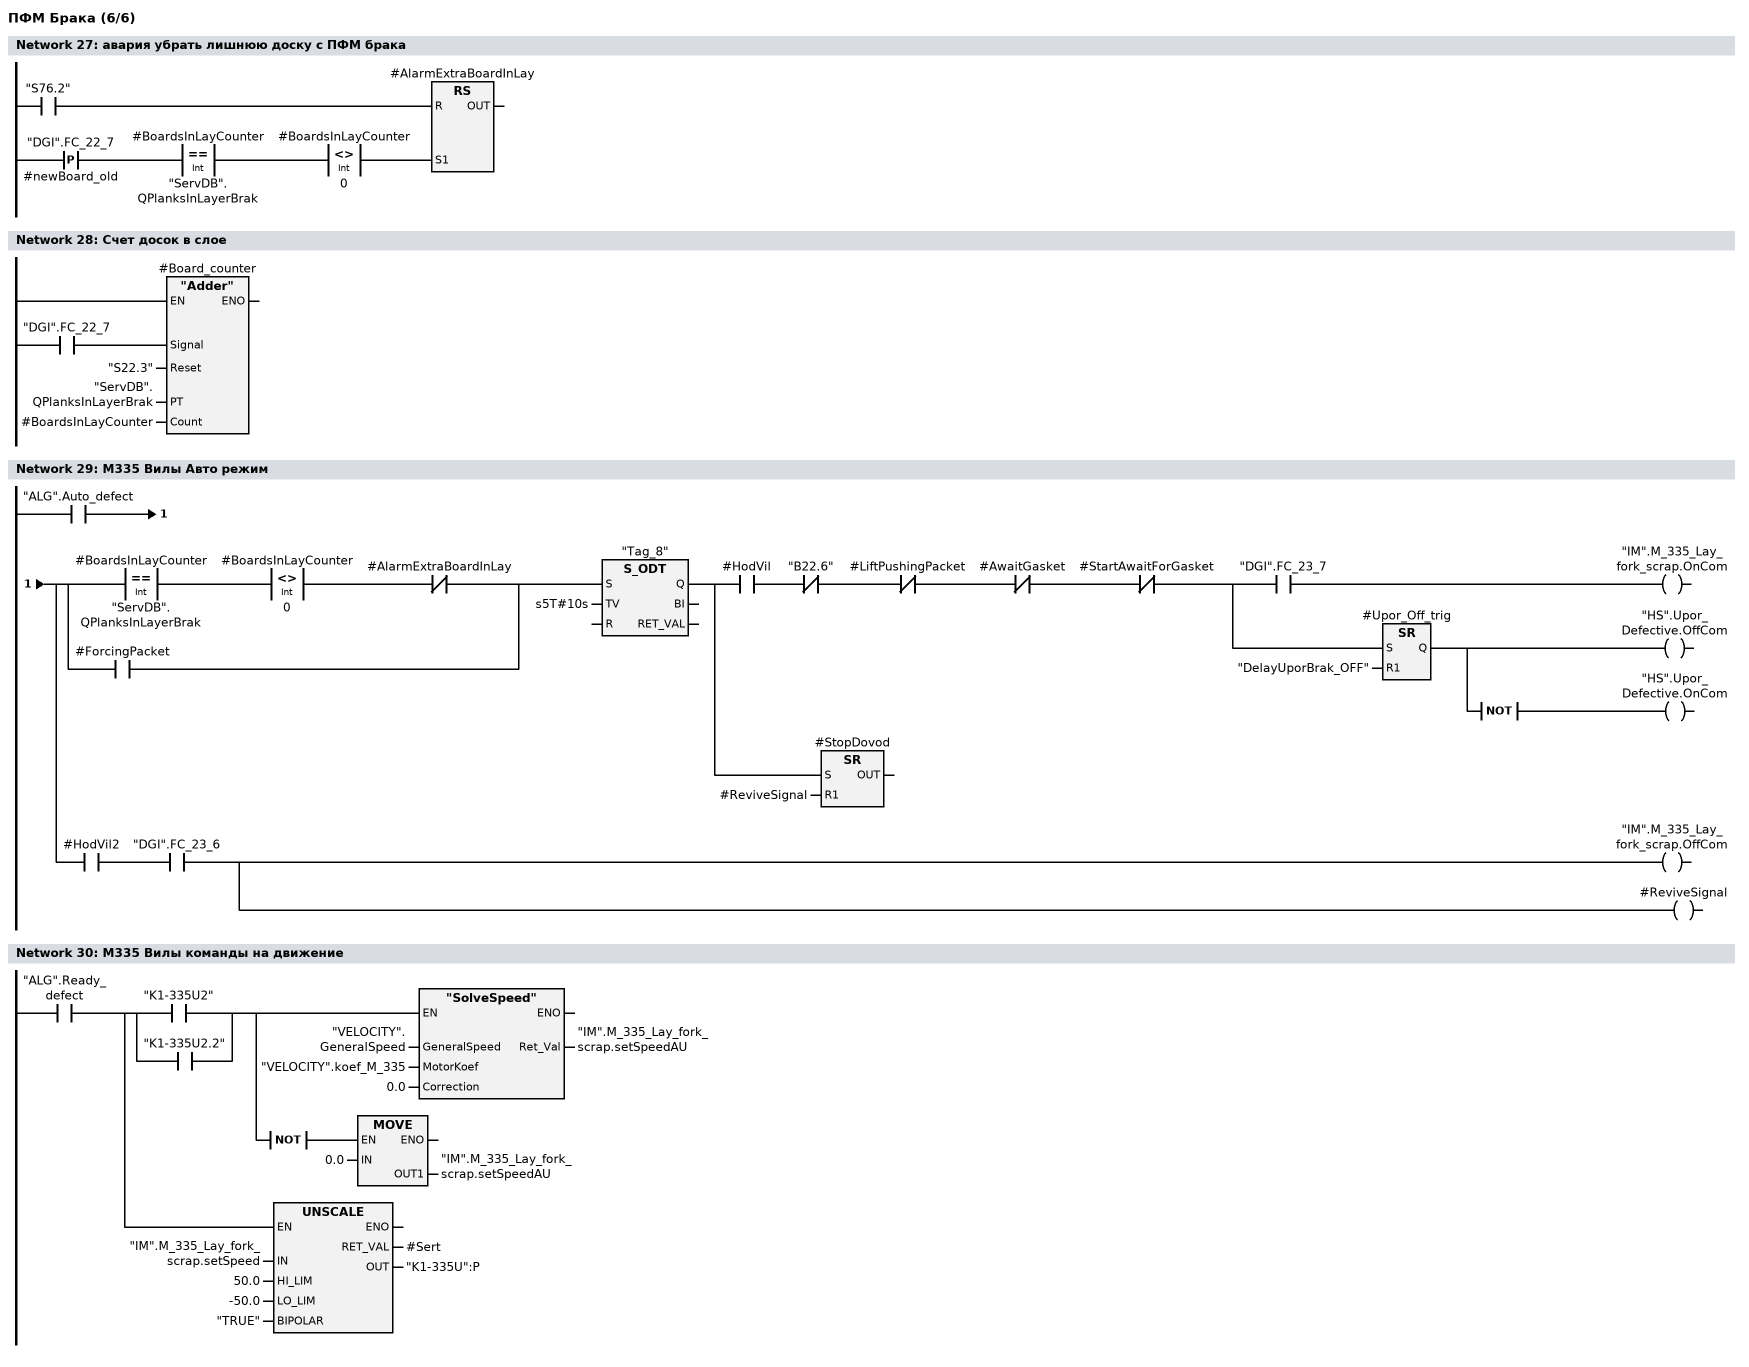
   RUNG wire#powerrail
      Contact( "S76.2" )
      S_RS(operand := #AlarmExtraBoardInLay, s1 := wire#w1)
   END_RUNG
   RUNG wire#powerrail
      P_Contact(operand := "DGI".FC_22_7, bit := #newBoard_old)
      { S7_Templates := "SrcType := Int" } EQ_Contact(in1 := #BoardsInLayCounter, in2 := "ServDB".QPlanksInLayerBrak)
      { S7_Templates := "SrcType := Int" } NE_Contact(in1 := #BoardsInLayCounter, in2 := 0)
   END_RUNG wire#w1
   // the same network as SCL:
   #_w1 := "DGI".FC_22_7 AND NOT #newBoard_old;   // rising edge of "DGI".FC_22_7
   #newBoard_old := "DGI".FC_22_7;
   IF "S76.2" THEN
       #AlarmExtraBoardInLay := FALSE;   // RS flip-flop
   END_IF;
   IF #_w1 AND (#BoardsInLayCounter = "ServDB".QPlanksInLayerBrak) AND (#BoardsInLayCounter <> 0) THEN
       #AlarmExtraBoardInLay := TRUE;
   END_IF;
END_REGION

REGION Network 28: Счет досок в слое
   RUNG wire#powerrail
      #Board_counter(Signal := wire#w1, Reset := "S22.3", PT := "ServDB".QPlanksInLayerBrak, Count := #BoardsInLayCounter)
   END_RUNG
   RUNG wire#powerrail
      Contact( "DGI".FC_22_7 )
   END_RUNG wire#w1
   // the same network as SCL:
   #Board_counter(Signal := "DGI".FC_22_7,   // "Adder"
                  Reset := "S22.3",
                  PT := "ServDB".QPlanksInLayerBrak,
                  Count := #BoardsInLayCounter);
END_REGION

REGION Network 29: М335 Вилы Авто режим
   RUNG wire#powerrail
      Contact( "ALG".Auto_defect )
      wire#w1
      { S7_Templates := "SrcType := Int" } EQ_Contact(in1 := #BoardsInLayCounter, in2 := "ServDB".QPlanksInLayerBrak)
      { S7_Templates := "SrcType := Int" } NE_Contact(in1 := #BoardsInLayCounter, in2 := 0)
      I_Contact( #AlarmExtraBoardInLay )
      wire#w2
      S_ODT(T_NO := "Tag_8", TV := s5T#10s, R :=, BI =>, RET_VAL =>)
      wire#w3
      Contact( #HodVil )
      I_Contact( "B22.6" )
      I_Contact( #LiftPushingPacket )
      I_Contact( #AwaitGasket )
      I_Contact( #StartAwaitForGasket )
      wire#w4
      Contact( "DGI".FC_23_7 )
      Coil( "IM".M_335_Lay_fork_scrap.OnCom )
   END_RUNG
   RUNG wire#w1
      Contact( #ForcingPacket )
   END_RUNG wire#w2
   RUNG wire#w4
      S_SR(operand := #Upor_Off_trig, r1 := "DelayUporBrak_OFF")
      wire#w5
      Coil( "HS".Upor_Defective.OffCom )
   END_RUNG
   RUNG wire#w5
      Not()
      Coil( "HS".Upor_Defective.OnCom )
   END_RUNG
   RUNG wire#w3
      S_SR(operand := #StopDovod, r1 := #ReviveSignal)
   END_RUNG
   RUNG wire#w1
      Contact( #HodVil2 )
      Contact( "DGI".FC_23_6 )
      wire#w6
      Coil( "IM".M_335_Lay_fork_scrap.OffCom )
   END_RUNG
   RUNG wire#w6
      Coil( #ReviveSignal )
   END_RUNG
   // the same network as SCL:
   #_w2 := "ALG".Auto_defect;
   #_s5time1 := S_ODT(T_NO := "Tag_8",
                      S := "ALG".Auto_defect AND (((#BoardsInLayCounter = "ServDB".QPlanksInLayerBrak) AND (#BoardsInLayCounter <> 0) AND NOT #AlarmExtraBoardInLay) OR #ForcingPacket),
                      TV := s5T#10s,
                      Q => #_w1);
   #_w3 := #_w1 AND #HodVil AND NOT "B22.6" AND NOT #LiftPushingPacket AND NOT #AwaitGasket AND NOT #StartAwaitForGasket;
   "IM".M_335_Lay_fork_scrap.OnCom := #_w3 AND "DGI".FC_23_7;
   IF #_w3 THEN
       #Upor_Off_trig := TRUE;   // SR flip-flop
   END_IF;
   IF "DelayUporBrak_OFF" THEN #Upor_Off_trig := FALSE; END_IF;
   "HS".Upor_Defective.OffCom := #Upor_Off_trig;
   "HS".Upor_Defective.OnCom := NOT #Upor_Off_trig;
   IF #_w1 THEN
       #StopDovod := TRUE;   // SR flip-flop
   END_IF;
   IF #ReviveSignal THEN #StopDovod := FALSE; END_IF;
   "IM".M_335_Lay_fork_scrap.OffCom := #_w2 AND #HodVil2 AND "DGI".FC_23_6;
   #ReviveSignal := "IM".M_335_Lay_fork_scrap.OffCom;
END_REGION

REGION Network 30: М335 Вилы команды на движение
   RUNG wire#powerrail
      Contact( "ALG".Ready_defect )
      wire#w1
      Contact( "K1-335U2" )
      wire#w2
      "SolveSpeed"(GeneralSpeed := "VELOCITY".GeneralSpeed, MotorKoef := "VELOCITY".koef_M_335, Correction := 0.0, Ret_Val => "IM".M_335_Lay_fork_scrap.setSpeedAU)
   END_RUNG
   RUNG wire#w1
      Contact( "K1-335U2.2" )
   END_RUNG wire#w2
   RUNG wire#w2
      Not()
      { S7_GenerateENO := "TRUE" } Move(in := 0.0, out1 => "IM".M_335_Lay_fork_scrap.setSpeedAU)
   END_RUNG
   RUNG wire#w1
      UNSCALE(IN := "IM".M_335_Lay_fork_scrap.setSpeed, HI_LIM := 50.0, LO_LIM := -50.0, BIPOLAR := "TRUE", RET_VAL => #Sert, OUT => "K1-335U":P)
   END_RUNG
   // the same network as SCL:
   #_w1 := "ALG".Ready_defect AND ("K1-335U2" OR "K1-335U2.2");
   #_w2 := "ALG".Ready_defect;
   IF #_w1 THEN
       "IM".M_335_Lay_fork_scrap.setSpeedAU := "SolveSpeed"(GeneralSpeed := "VELOCITY".GeneralSpeed,
                               MotorKoef := "VELOCITY".koef_M_335,
                               Correction := 0.0);
   END_IF;
   IF NOT #_w1 THEN "IM".M_335_Lay_fork_scrap.setSpeedAU := 0.0; END_IF;
   IF #_w2 THEN
       #Sert := UNSCALE(IN := "IM".M_335_Lay_fork_scrap.setSpeed,
                        HI_LIM := 50.0,
                        LO_LIM := -50.0,
                        BIPOLAR := "TRUE",
                        OUT => "K1-335U":P);
   END_IF;
END_REGION
END_FUNCTION_BLOCK
